// Mitsubishi GX Works2 project: jump   PLC: Q03UDV

PROGRAM MAIN
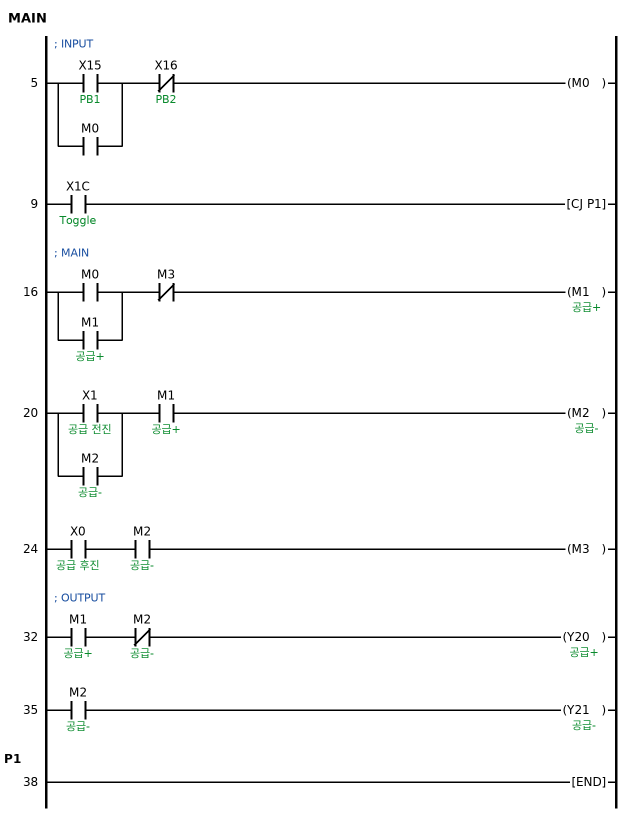
; INPUT
5     LD      X15  ; PB1
      OR      M0
      ANI     X16  ; PB2
      OUT     M0
9     LD      X1C  ; Toggle
      CJ      P1  ; STOP
; MAIN
16    LD      M0
      OR      M1  ; 공급+
      ANI     M3
      OUT     M1  ; 공급+
20    LD      X1  ; 공급 전진
      OR      M2  ; 공급-
      AND     M1  ; 공급+
      OUT     M2  ; 공급-
24    LD      X0  ; 공급 후진
      AND     M2  ; 공급-
      OUT     M3
; OUTPUT
32    LD      M1  ; 공급+
      ANI     M2  ; 공급-
      OUT     Y20  ; 공급+
35    LD      M2  ; 공급-
      OUT     Y21  ; 공급-
      P1
38    END
END_PROGRAM
